FUNCTION_BLOCK AX_TO_AQ (* Converts an AX (BOOL) adapter to an AQ (Quarter Byte) adapter using COMMAND logic *)
  (* Standard: 61499-2; Description: Copyright (c) 2026 Meisterschulen am Ostbahnhof SPDX-License-Identifier: EPL-2.0 *)
  (* Version 1.0, 2026-05-16, Franz Höpfinger, Meisterschulen am Ostbahnhof, Initial Version *)
  PACKAGE adapter::conversion::unidirectional;
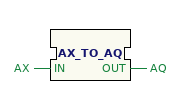
  SOCKETS
    IN : adapter::types::unidirectional::AX; (* BOOL Input *)
  END_SOCKETS
  PLUGS
    OUT : adapter::types::unidirectional::AQ; (* AQ Output *)
  END_PLUGS
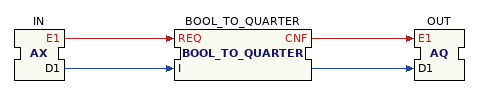
  FBS
    BOOL_TO_QUARTER : logiBUS::utils::quarter::BOOL_TO_QUARTER;
  END_FBS
  EVENT_CONNECTIONS
    IN.E1 TO BOOL_TO_QUARTER.REQ;
    BOOL_TO_QUARTER.CNF TO OUT.E1;
  END_CONNECTIONS
  DATA_CONNECTIONS
    IN.D1 TO BOOL_TO_QUARTER.I;
    BOOL_TO_QUARTER. TO OUT.D1;
  END_CONNECTIONS
END_FUNCTION_BLOCK
